TYPE ST_Chamber1VacuumOnParam :
STRUCT
END_STRUCT
END_TYPE

(* stored: Version 1.1.0.1, ProductVersion 3.1.4026.18
   DUT ST_Chamber1VacuumOnParam: Id {9aed5ace-5700-4979-b77b-58334c2eb308} *)
